// TIA Portal V17 export
// export: Created 2025-03-10T13:12:35.1156182Z, ExportSetting WithDefaults, DisplayName Totally Integrated Automation Portal, DisplayVersion V17 Update 8, DisplayName TIA Portal Openness, DisplayVersion V17 Update 8, DisplayName TIA Portal Version Control Interface, DisplayVersion V17, DisplayName SINAMICS Startdrive Advanced, DisplayVersion V17 SP2, DisplayName SINAMICS Startdrive G110M, G120, G120C, G120D, G120P, G115D, DisplayVersion V17 SP2, DisplayName SINAMICS Startdrive G130, G150, S120, S150, SINAMICS MV, S210, DisplayVersion V17 SP2, DisplayName STEP 7 Professional, DisplayVersion V17 Update 8, DisplayName SINUMERIK ONE STEP 7 Toolbox, DisplayVersion V17 Update 12, DisplayName SINUMERIK 840D sl STEP 7 Toolbox, DisplayVersion V17 Update 12, DisplayName STEP 7 Safety, DisplayVersion V17 Update 6, DisplayName WinCC Advanced, DisplayVersion V17 Update 8
FUNCTION "FC2121_MPP" : Void   // FC2121, LAD
{ S7_Optimized_Access := 'FALSE' }
AUTHOR : ETXETAR
VERSION : 1.0
// stored: AutoNumber false, IsIECCheckEnabled false, SetENOAutomatically false, UDAEnableTagReadback false
   VAR_TEMP
      ONE : Int;
      RETVAL1 : Int;
      SIMU_PANEL_HMI_SEL : Bool;   // SIMULATED PANEL IN HMI SELECTED
   END_VAR
   VAR CONSTANT
      FC_NUMBER : DInt := 2121;   // FC NUMBER
   END_VAR
BEGIN

REGION Network 1: INPUTS
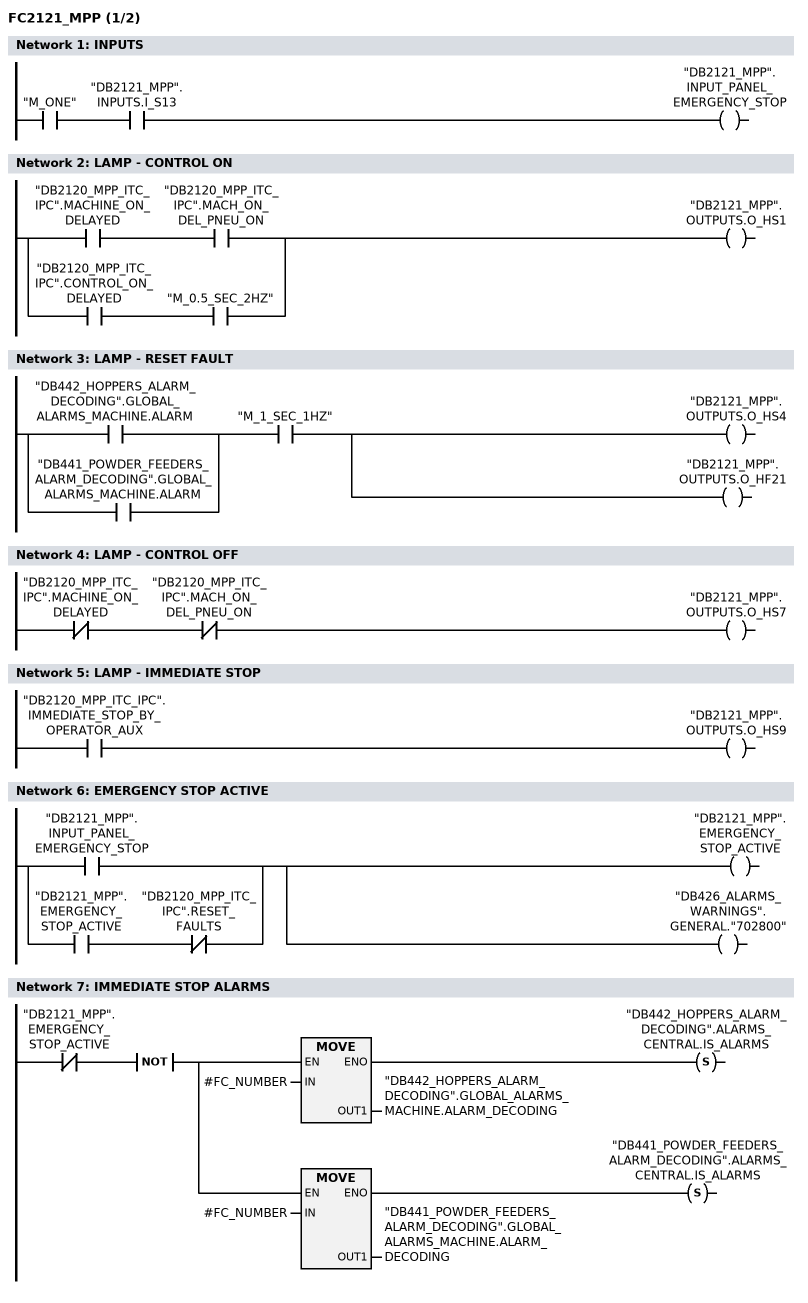
   RUNG wire#powerrail
      Contact( "M_ONE" )
      Contact( "DB2121_MPP".INPUTS.I_S13 )
      Coil( "DB2121_MPP".INPUT_PANEL_EMERGENCY_STOP )
   END_RUNG
   // the same network as SCL:
   "DB2121_MPP".INPUT_PANEL_EMERGENCY_STOP := "M_ONE" AND "DB2121_MPP".INPUTS.I_S13;
END_REGION

REGION Network 2: LAMP - CONTROL ON
   RUNG wire#powerrail
      Contact( "DB2120_MPP_ITC_IPC".MACHINE_ON_DELAYED )
      Contact( "DB2120_MPP_ITC_IPC".MACH_ON_DEL_PNEU_ON )
      wire#w1
      Coil( "DB2121_MPP".OUTPUTS.O_HS1 )
   END_RUNG
   RUNG wire#powerrail
      Contact( "DB2120_MPP_ITC_IPC".CONTROL_ON_DELAYED )
      Contact( "M_0.5_SEC_2HZ" )
   END_RUNG wire#w1
   // the same network as SCL:
   "DB2121_MPP".OUTPUTS.O_HS1 := ("DB2120_MPP_ITC_IPC".MACHINE_ON_DELAYED AND "DB2120_MPP_ITC_IPC".MACH_ON_DEL_PNEU_ON) OR ("DB2120_MPP_ITC_IPC".CONTROL_ON_DELAYED AND "M_0.5_SEC_2HZ");
END_REGION

REGION Network 3: LAMP - RESET FAULT
   RUNG wire#powerrail
      Contact( "DB442_HOPPERS_ALARM_DECODING".GLOBAL_ALARMS_MACHINE.ALARM )
      wire#w1
      Contact( "M_1_SEC_1HZ" )
      wire#w2
      Coil( "DB2121_MPP".OUTPUTS.O_HS4 )
   END_RUNG
   RUNG wire#powerrail
      Contact( "DB441_POWDER_FEEDERS_ALARM_DECODING".GLOBAL_ALARMS_MACHINE.ALARM )
   END_RUNG wire#w1
   RUNG wire#w2
      Coil( "DB2121_MPP".OUTPUTS.O_HF21 )
   END_RUNG
   // the same network as SCL:
   "DB2121_MPP".OUTPUTS.O_HS4 := ("DB442_HOPPERS_ALARM_DECODING".GLOBAL_ALARMS_MACHINE.ALARM OR "DB441_POWDER_FEEDERS_ALARM_DECODING".GLOBAL_ALARMS_MACHINE.ALARM) AND "M_1_SEC_1HZ";
   "DB2121_MPP".OUTPUTS.O_HF21 := "DB2121_MPP".OUTPUTS.O_HS4;
END_REGION

REGION Network 4: LAMP - CONTROL OFF
   RUNG wire#powerrail
      I_Contact( "DB2120_MPP_ITC_IPC".MACHINE_ON_DELAYED )
      I_Contact( "DB2120_MPP_ITC_IPC".MACH_ON_DEL_PNEU_ON )
      Coil( "DB2121_MPP".OUTPUTS.O_HS7 )
   END_RUNG
   // the same network as SCL:
   "DB2121_MPP".OUTPUTS.O_HS7 := NOT "DB2120_MPP_ITC_IPC".MACHINE_ON_DELAYED AND NOT "DB2120_MPP_ITC_IPC".MACH_ON_DEL_PNEU_ON;
END_REGION

REGION Network 5: LAMP - IMMEDIATE STOP
   RUNG wire#powerrail
      Contact( "DB2120_MPP_ITC_IPC".IMMEDIATE_STOP_BY_OPERATOR_AUX )
      Coil( "DB2121_MPP".OUTPUTS.O_HS9 )
   END_RUNG
   // the same network as SCL:
   "DB2121_MPP".OUTPUTS.O_HS9 := "DB2120_MPP_ITC_IPC".IMMEDIATE_STOP_BY_OPERATOR_AUX;
END_REGION

REGION Network 6: EMERGENCY STOP ACTIVE
   RUNG wire#powerrail
      Contact( "DB2121_MPP".INPUT_PANEL_EMERGENCY_STOP )
      wire#w1
      Coil( "DB2121_MPP".EMERGENCY_STOP_ACTIVE )
   END_RUNG
   RUNG wire#powerrail
      Contact( "DB2121_MPP".EMERGENCY_STOP_ACTIVE )
      I_Contact( "DB2120_MPP_ITC_IPC".RESET_FAULTS )
   END_RUNG wire#w1
   RUNG wire#w1
      Coil( "DB426_ALARMS_WARNINGS".GENERAL."702800" )
   END_RUNG
   // the same network as SCL:
   "DB2121_MPP".EMERGENCY_STOP_ACTIVE := "DB2121_MPP".INPUT_PANEL_EMERGENCY_STOP OR ("DB2121_MPP".EMERGENCY_STOP_ACTIVE AND NOT "DB2120_MPP_ITC_IPC".RESET_FAULTS);
   "DB426_ALARMS_WARNINGS".GENERAL."702800" := "DB2121_MPP".EMERGENCY_STOP_ACTIVE;
END_REGION

REGION Network 7: IMMEDIATE STOP ALARMS
   RUNG wire#powerrail
      I_Contact( "DB2121_MPP".EMERGENCY_STOP_ACTIVE )
      Not()
      wire#w1
      { S7_GenerateENO := "TRUE" } Move(in := #FC_NUMBER, out1 => "DB442_HOPPERS_ALARM_DECODING".GLOBAL_ALARMS_MACHINE.ALARM_DECODING)
      S_Coil( "DB442_HOPPERS_ALARM_DECODING".ALARMS_CENTRAL.IS_ALARMS )
   END_RUNG
   RUNG wire#w1
      { S7_GenerateENO := "TRUE" } Move(in := #FC_NUMBER, out1 => "DB441_POWDER_FEEDERS_ALARM_DECODING".GLOBAL_ALARMS_MACHINE.ALARM_DECODING)
      S_Coil( "DB441_POWDER_FEEDERS_ALARM_DECODING".ALARMS_CENTRAL.IS_ALARMS )
   END_RUNG
   // the same network as SCL:
   // ENO of a box is taken as its EN; it also drops when the box reports an error
   IF NOT (NOT "DB2121_MPP".EMERGENCY_STOP_ACTIVE) THEN
       "DB442_HOPPERS_ALARM_DECODING".GLOBAL_ALARMS_MACHINE.ALARM_DECODING := #FC_NUMBER;
       "DB442_HOPPERS_ALARM_DECODING".ALARMS_CENTRAL.IS_ALARMS := TRUE;
       "DB441_POWDER_FEEDERS_ALARM_DECODING".GLOBAL_ALARMS_MACHINE.ALARM_DECODING := #FC_NUMBER;
       "DB441_POWDER_FEEDERS_ALARM_DECODING".ALARMS_CENTRAL.IS_ALARMS := TRUE;
   END_IF;
END_REGION

REGION Network 8: WARNING
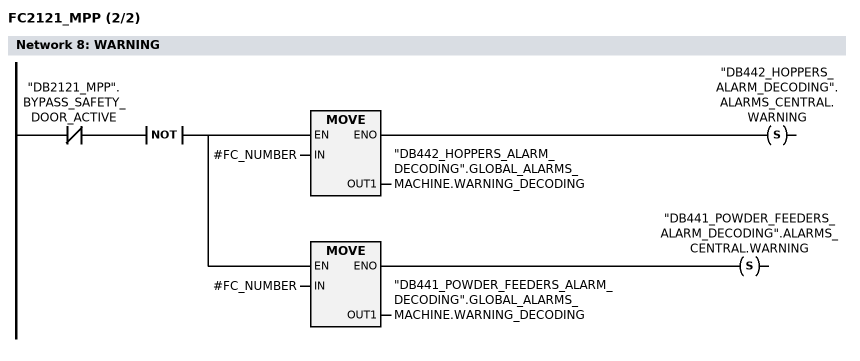
   RUNG wire#powerrail
      I_Contact( "DB2121_MPP".BYPASS_SAFETY_DOOR_ACTIVE )
      Not()
      wire#w1
      { S7_GenerateENO := "TRUE" } Move(in := #FC_NUMBER, out1 => "DB442_HOPPERS_ALARM_DECODING".GLOBAL_ALARMS_MACHINE.WARNING_DECODING)
      S_Coil( "DB442_HOPPERS_ALARM_DECODING".ALARMS_CENTRAL.WARNING )
   END_RUNG
   RUNG wire#w1
      { S7_GenerateENO := "TRUE" } Move(in := #FC_NUMBER, out1 => "DB441_POWDER_FEEDERS_ALARM_DECODING".GLOBAL_ALARMS_MACHINE.WARNING_DECODING)
      S_Coil( "DB441_POWDER_FEEDERS_ALARM_DECODING".ALARMS_CENTRAL.WARNING )
   END_RUNG
   // the same network as SCL:
   // ENO of a box is taken as its EN; it also drops when the box reports an error
   IF NOT (NOT "DB2121_MPP".BYPASS_SAFETY_DOOR_ACTIVE) THEN
       "DB442_HOPPERS_ALARM_DECODING".GLOBAL_ALARMS_MACHINE.WARNING_DECODING := #FC_NUMBER;
       "DB442_HOPPERS_ALARM_DECODING".ALARMS_CENTRAL.WARNING := TRUE;
       "DB441_POWDER_FEEDERS_ALARM_DECODING".GLOBAL_ALARMS_MACHINE.WARNING_DECODING := #FC_NUMBER;
       "DB441_POWDER_FEEDERS_ALARM_DECODING".ALARMS_CENTRAL.WARNING := TRUE;
   END_IF;
END_REGION
END_FUNCTION
